(* CODESYS project CtaAppBasic_1.0.0.1.library
   Description: Basic Library der CTA
   Version: 1.0.0.1
   Title: CtaAppBasic
   Author: SIS
   DocFormat: reStructuredText
   LanguageModelAttribute: qualified-access-only
   Placeholder: CtaAppBasic
   DefaultNamespace: CtaAppBasic
   CompiledLibraryCompatibilityVersion: CODESYS V3.5 SP16 Patch 3
   Company: CTA

Project tree, tasks and I/O mapping:
  libraries: VisuSymbols, 4.5.0.0 (System); Standard, 3.5.18.0 (System); CtaAppTime, 1.0.0.1 (CTA)
  40 Visualizations/
  30 Program Organization Units/
    SCALER/
      function fcScale [ST]
      function block fbscaleDreifach [ST]
      function block fbscaleVierfach [ST]
    AVERAGE/
      function block fbAverageAt [ST]: GetAverageAT
  00000000-0000-0000-0000-000000000000|D:\CoDeSys\LibrariesV3\trunk\Intern\CAA\CAA Template\3.4.0.0 draft\Placeholder.xml
  00000000-0000-0000-0000-000000000000|D:\CoDeSys\LibrariesV3\trunk\Intern\CAA\CAA Template\3.2.0.3 draft\Prefix.pdf
  00000000-0000-0000-0000-000000000000|D:\CoDeSys\LibrariesV3\trunk\Intern\CAA\CAA Template\3.5.2.0 draft\Placeholder.xml
  20 Structs/
  50 Images/
  10 Documenation/
    global variables VersionHistory
    global variables readMe
  21 Interface/
  11 Library Parameter/
  12 Konstanten/
  60 Textlisten/
  13 Globale Variablen/
*)

// 10 Documenation/VersionHistory
(* 

.. image:: ../../Images/CTA_Logo.jpg
   :align: right
   :width: 15% 

**Vorlage**   


============ =========== =========== ============================================
**Date**     **Version** **Author**  **Change**
------------ ----------- ----------- --------------------------------------------
04.03.2021   0.0.0.0     SIS         Vorlage erstellt

============ =========== =========== ============================================


*)
VAR_GLOBAL
    stInfo : STRING:= '0.0.0.0, Vorlage, CTA';
END_VAR

// 10 Documenation/readMe
(*

**ReadMe**
 
|	**Empfehlung**
|
|	Dokumentrieren Sie die Library für eine nachhaltige Entwicklung
|     
| *Beispiel* 
|
| Dies ist die Vorlage Library der CTA. Erstellen Sie ihre Library anhand dieser Vorlage.
*)

VAR_GLOBAL
    xReadMeDone              :   BOOL;
END_VAR

// 30 Program Organization Units/SCALER/fcScale
FUNCTION fcScale : REAL
VAR_INPUT
    rIn          :  REAL;
    rMin         :  REAL;
    rMax         :  REAL;
    rOutMin      :  REAL;
    rOutMax      :  REAL;
END_VAR
VAR
END_VAR

fcScale := (((rIn - rMin)*(rOutMax - rOutMin)) / SEL(rMin <> rMax,1,(rMax-rMin))) + rOutMin;

END_FUNCTION

// 30 Program Organization Units/SCALER/fbscaleDreifach
FUNCTION_BLOCK fbscaleDreifach
(*
Erklärung:
1. Flag für aufsteigende X-Achse (ascendingX): Bestimmt, ob die X-Werte aufsteigend sind oder nicht.
2. Min- und Max-Werte: Berechnet die minimalen und maximalen X- und Y-Werte.
3. Interpolation und Abfangen:
	- Wenn die X-Achse aufsteigend ist, wird der output entsprechend interpoliert oder auf den minimalen/maximalen Y-Wert gesetzt, wenn input außerhalb des Bereichs liegt.
	- Wenn die X-Achse absteigend ist, wird ebenfalls interpoliert oder die Grenzwerte verwendet.
	
Funktionsweise:
Das Programm berücksichtigt sowohl aufsteigende als auch absteigende X-Achsen-Werte und interpoliert oder setzt den output entsprechend der Position von input innerhalb oder außerhalb der definierten X-Werte. 
Es stellt sicher, dass die output-Werte innerhalb der definierten Min- und Max-Grenzen liegen.*)

VAR_INPUT
	rInput 		: REAL;                      // Eingabewert
	
	x1			: REAL;
	x2			: REAL;
	x3			: REAL;
	y1			: REAL;
	y2			: REAL;
	y3			: REAL;
END_VAR
VAR_OUTPUT
	rOutput 	: REAL;           // Ausgabewert (kann Y oder X sein)
END_VAR
VAR
	xAxis : ARRAY[1..3] OF REAL;  // X-Achsen-Werte
    yAxis : ARRAY[1..3] OF REAL;  // Y-Achsen-Werte
    
    i : INT;                            // Schleifenindex
    slope : REAL;                       // Steigung zwischen zwei Punkten
    xMin, xMax : REAL;                  // Minimaler und maximaler X-Wert
    yMin, yMax : REAL;                  // Minimaler und maximaler Y-Wert
    ascendingX : BOOL;                  // Flag für aufsteigende X-Achse
    intervalFound : BOOL := FALSE;      // Flag, ob das richtige Intervall gefunden wurde
END_VAR

// Initialisierung der X- und Y-Achsen-Werte
xAxis[1] := x1;
xAxis[2] := x2;
xAxis[3] := x3;

yAxis[1] := y1;
yAxis[2] := y2;
yAxis[3] := y3;

// Bestimme, ob die X-Achse aufsteigend ist
ascendingX := xAxis[1] < xAxis[2];

// Bestimme Min- und Max-Werte der X- und Y-Achse
xMin := MIN(xAxis[1], MIN(xAxis[2],xAxis[3]));
xMax := MAX(xAxis[1], MAX(xAxis[2],xAxis[3]));

yMin := MIN(yAxis[1], MIN(yAxis[2],yAxis[3]));
yMax := MAX(yAxis[1], MAX(yAxis[2],yAxis[3]));

// Interpolation oder Abfanglogik
IF ascendingX THEN
    // X-Achse ist aufsteigend
    IF rInput <= xMin THEN
        rOutput := yAxis[1];
    ELSIF rInput >= xMax THEN
        rOutput := yAxis[3];
    ELSE
        FOR i := 1 TO 2 DO
            IF (xAxis[i] <= rInput) AND (rInput <= xAxis[i+1]) THEN
                slope := (yAxis[i+1] - yAxis[i]) / (xAxis[i+1] - xAxis[i]);
                rOutput := yAxis[i] + slope * (rInput - xAxis[i]);
                intervalFound := TRUE;
                EXIT;
            END_IF;
        END_FOR
        // Falls kein Intervall gefunden wurde
        IF NOT intervalFound THEN
            rOutput := yAxis[3];
        END_IF;
    END_IF;
ELSE
    // X-Achse ist absteigend
    IF rInput >= xMax THEN
        rOutput := yAxis[1];
    ELSIF rInput <= xMin THEN
        rOutput := yAxis[3];
    ELSE
        FOR i := 1 TO 2 DO
            IF (xAxis[i] >= rInput) AND (rInput >= xAxis[i+1]) THEN
                slope := (yAxis[i+1] - yAxis[i]) / (xAxis[i+1] - xAxis[i]);
                rOutput := yAxis[i] + slope * (rInput - xAxis[i]);
                intervalFound := TRUE;
                EXIT;
            END_IF;
        END_FOR
        // Falls kein Intervall gefunden wurde
        IF NOT intervalFound THEN
            rOutput := yAxis[3];
        END_IF;
    END_IF;
END_IF

END_FUNCTION_BLOCK

// 30 Program Organization Units/SCALER/fbscaleVierfach
FUNCTION_BLOCK fbscaleVierfach
(*
Erklärung:
1. Flag für aufsteigende X-Achse (ascendingX): Bestimmt, ob die X-Werte aufsteigend sind oder nicht.
2. Min- und Max-Werte: Berechnet die minimalen und maximalen X- und Y-Werte.
3. Interpolation und Abfangen:
	- Wenn die X-Achse aufsteigend ist, wird der output entsprechend interpoliert oder auf den minimalen/maximalen Y-Wert gesetzt, wenn input außerhalb des Bereichs liegt.
	- Wenn die X-Achse absteigend ist, wird ebenfalls interpoliert oder die Grenzwerte verwendet.
	
Funktionsweise:
Das Programm berücksichtigt sowohl aufsteigende als auch absteigende X-Achsen-Werte und interpoliert oder setzt den output entsprechend der Position von input innerhalb oder außerhalb der definierten X-Werte. 
Es stellt sicher, dass die output-Werte innerhalb der definierten Min- und Max-Grenzen liegen.*)

VAR_INPUT
	rInput 		: REAL;                      // Eingabewert
	
	x1			: REAL;
	x2			: REAL;
	x3			: REAL;
	x4			: REAL;	
	y1			: REAL;
	y2			: REAL;
	y3			: REAL;
	y4			: REAL;
END_VAR
VAR_OUTPUT
	rOutput 	: REAL;           // Ausgabewert (kann Y oder X sein)
END_VAR
VAR
	xAxis : ARRAY[1..4] OF REAL;  // X-Achsen-Werte
    yAxis : ARRAY[1..4] OF REAL;  // Y-Achsen-Werte
    
    i : INT;                            // Schleifenindex
    slope : REAL;                       // Steigung zwischen zwei Punkten
    xMin, xMax : REAL;                  // Minimaler und maximaler X-Wert
    yMin, yMax : REAL;                  // Minimaler und maximaler Y-Wert
    ascendingX : BOOL;                  // Flag für aufsteigende X-Achse
    intervalFound : BOOL := FALSE;      // Flag, ob das richtige Intervall gefunden wurde
END_VAR

// Initialisierung der X- und Y-Achsen-Werte
xAxis[1] := x1;
xAxis[2] := x2;
xAxis[3] := x3;
xAxis[4] := x4;

yAxis[1] := y1;
yAxis[2] := y2;
yAxis[3] := y3;
yAxis[4] := y4;

// Bestimme, ob die X-Achse aufsteigend ist
ascendingX := xAxis[1] < xAxis[2];

// Bestimme Min- und Max-Werte der X- und Y-Achse
xMin := MIN(xAxis[1], MIN(xAxis[2], MIN(xAxis[3], xAxis[4])));
xMax := MAX(xAxis[1], MAX(xAxis[2], MAX(xAxis[3], xAxis[4])));

yMin := MIN(yAxis[1], MIN(yAxis[2], MIN(yAxis[3], yAxis[4])));
yMax := MAX(yAxis[1], MAX(yAxis[2], MAX(yAxis[3], yAxis[4])));

// Interpolation oder Abfanglogik
IF ascendingX THEN
    // X-Achse ist aufsteigend
    IF rInput <= xMin THEN
        rOutput := yAxis[1];
    ELSIF rInput >= xMax THEN
        rOutput := yAxis[4];
    ELSE
        FOR i := 1 TO 3 DO
            IF (xAxis[i] <= rInput) AND (rInput <= xAxis[i+1]) THEN
                slope := (yAxis[i+1] - yAxis[i]) / (xAxis[i+1] - xAxis[i]);
                rOutput := yAxis[i] + slope * (rInput - xAxis[i]);
                intervalFound := TRUE;
                EXIT;
            END_IF;
        END_FOR
        // Falls kein Intervall gefunden wurde
        IF NOT intervalFound THEN
            rOutput := yAxis[4];
        END_IF;
    END_IF;
ELSE
    // X-Achse ist absteigend
    IF rInput >= xMax THEN
        rOutput := yAxis[1];
    ELSIF rInput <= xMin THEN
        rOutput := yAxis[4];
    ELSE
        FOR i := 1 TO 3 DO
            IF (xAxis[i] >= rInput) AND (rInput >= xAxis[i+1]) THEN
                slope := (yAxis[i+1] - yAxis[i]) / (xAxis[i+1] - xAxis[i]);
                rOutput := yAxis[i] + slope * (rInput - xAxis[i]);
                intervalFound := TRUE;
                EXIT;
            END_IF;
        END_FOR
        // Falls kein Intervall gefunden wurde
        IF NOT intervalFound THEN
            rOutput := yAxis[4];
        END_IF;
    END_IF;
END_IF

END_FUNCTION_BLOCK

// 30 Program Organization Units/AVERAGE/fbAverageAt
FUNCTION_BLOCK fbAverageAt 
VAR_INPUT
	rAT	:	REAL;
END_VAR
VAR
	ayMesurement	:	ARRAY[0..719] OF REAL;
	ayMesurementDt	:	ARRAY[0..719] OF DT;
	Trig			:	TON;
	Index			:	INT;
	Intervall		:	TIME	:= T#2m;
END_VAR

Trig(in := NOT trig.Q,PT:= Intervall);

IF Index >= 719 THEN 
	index := 0;
END_IF;
IF Trig.Q THEN
	ayMesurement[Index] := rAT;
	ayMesurementDt[Index] := CtaAppTime.FuGetLocalDateAndTime();
	Index := Index + 1;
END_IF

METHOD GetAverageAT : REAL
VAR_INPUT
	TimeRange	:	TIME;
END_VAR
VAR
	TimeRangeAsDt	:	DT;
	CurrentDt		:	DT;
	i				:	INT;
	count			:	INT;
	rAtSumme		:	REAL;
END_VAR
TimeRangeAsDt := TO_DT(MIN(TimeRange,T#24H));
CurrentDt := CtaAppTime.FuGetLocalDateAndTime();

FOR i:= 0 TO 719 DO 
	IF ayMesurementDt[i] >= TO_DT(CurrentDt - TimeRangeAsDt) THEN
		rAtSumme := rAtSumme + ayMesurement[i];
		count := count + 1;
		GetAverageAT := rAtSumme / count;
	END_IF;
END_FOR;
END_METHOD

END_FUNCTION_BLOCK
